// TIA Portal V21 export
VAR_GLOBAL   // PLC tag table "K_TipoMacchina"
END_VAR
VAR_GLOBAL CONSTANT   // user constants
   K_TipoMacchina_Pastorizzatore : Int := 0;
   K_TipoMacchina_ProcessoGenerico : Int := 1;
   K_TipoMacchina_Trasporti : Int := 2;
   K_TipoMacchina_Pallettizzatore : Int := 3;
   K_TipoMacchina_Depallettizzatore : Int := 4;
END_VAR
